ABB RobotStudio station: Project_Lab2.rsstnx

Station Project1 (saved by RobotStudio 25.1.11167.1)
Controller Controller_Lab2
  mechanical unit ROB_1: IRB140_6_81_C_03, 6 joints, base frame (0, 0, 0) mm
Layout (positions relative to the parent item):
  - IRB140_6_81_C_03 [mechanism, from %ABB.RobotStudio.Models.IRB140%\IRB140_6_81_C_G_03.rslib] at (0, 0, 0) mm; joint values [-0.0202, 0.226, 0.2165, 0.0425, 0.3433, -0.0544] (rad or m)
  - Marcador_2 [mechanism, from Project_Lab2\Marcador.rslib] at (539.94, -10, 494.18) mm, rotated rx -180 ry 45 rz -180 deg
  - Pastel [part] at (500, 0, 250) mm, rotated rx 0 ry 0 rz -90 deg, size 272 x 195 x 20 mm
Attachment: Marcador_2 is attached to IRB140_6_81_C_03 / Link6
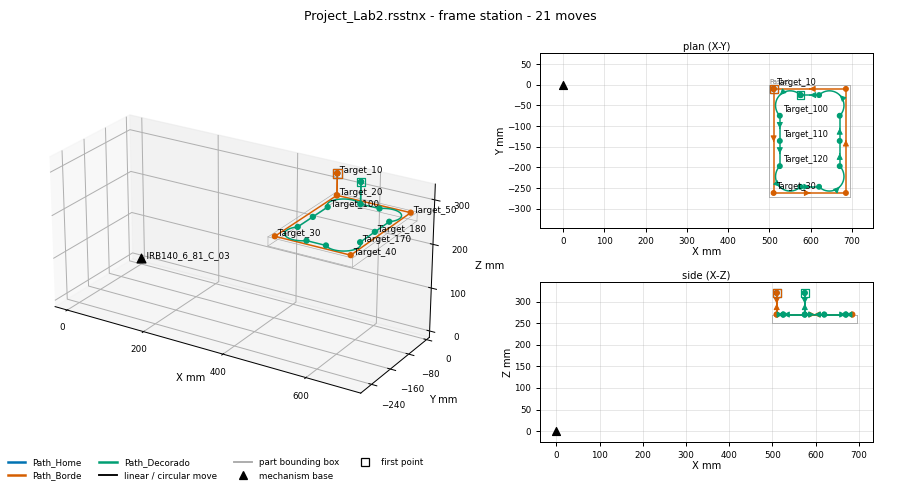
[picture p0: tool path of Project_Lab2.rsstnx in frame station, 21 of 21 moves have a stored position in this frame; points joined in program order, loops and branches not executed]
Targets, tools, work objects and paths stored in the station, written as RAPID:
! task T_ROB1
MODULE CalibData
  PERS tooldata TCP_Marcador:=[TRUE,[[144.332,0,101.99],[0.866025404,0,0.5,0]],[1,[0,0,1],[1,0,0,0],0,0,0]];
  TASK PERS wobjdata Workobject_pastel:=[FALSE,TRUE,"",[[500,0,250],[0.707106781,0,0,-0.707106781]],[[0,0,0],[1,0,0,0]]];
ENDMODULE

! task T_ROB1
MODULE Module1
  CONST robtarget Target_10:=[[10,10,70],[0.092295955,0.701057385,-0.701057385,0.092295955],[0,0,0,0],[9E+09,9E+09,9E+09,9E+09,9E+09,9E+09]];
  CONST robtarget Target_20:=[[10,10,20],[0.092295955,0.701057385,-0.701057385,0.092295955],[0,0,0,0],[9E+09,9E+09,9E+09,9E+09,9E+09,9E+09]];
  CONST robtarget Target_30:=[[262,10,20],[0.092295955,0.701057385,-0.701057385,0.092295955],[0,0,0,0],[9E+09,9E+09,9E+09,9E+09,9E+09,9E+09]];
  CONST robtarget Target_40:=[[262,185,20],[0.092295955,0.701057385,-0.701057385,0.092295955],[0,0,0,0],[9E+09,9E+09,9E+09,9E+09,9E+09,9E+09]];
  CONST robtarget Target_50:=[[10,185,20],[0.092295955,0.701057385,-0.701057385,0.092295955],[0,0,0,0],[9E+09,9E+09,9E+09,9E+09,9E+09,9E+09]];
  CONST robtarget Target_60:=[[10,10,20],[0.092295955,0.701057385,-0.701057385,0.092295955],[0,0,0,0],[9E+09,9E+09,9E+09,9E+09,9E+09,9E+09]];
  CONST robtarget Target_70:=[[25,75,70],[0.092295955,0.701057385,-0.701057385,0.092295955],[-1,0,-1,0],[9E+09,9E+09,9E+09,9E+09,9E+09,9E+09]];
  CONST robtarget Target_80:=[[25,75,20],[0.092295955,0.701057385,-0.701057385,0.092295955],[-1,0,-1,0],[9E+09,9E+09,9E+09,9E+09,9E+09,9E+09]];
  CONST robtarget Target_90:=[[25,25,20],[0.092295955,0.701057385,-0.701057385,0.092295955],[-1,0,-1,0],[9E+09,9E+09,9E+09,9E+09,9E+09,9E+09]];
  CONST robtarget Target_100:=[[75,25,20],[0.092295955,0.701057385,-0.701057385,0.092295955],[-1,0,-1,0],[9E+09,9E+09,9E+09,9E+09,9E+09,9E+09]];
  CONST robtarget Target_110:=[[136,25,20],[0.092295955,0.701057385,-0.701057385,0.092295955],[-1,0,-1,0],[9E+09,9E+09,9E+09,9E+09,9E+09,9E+09]];
  CONST robtarget Target_120:=[[197,25,20],[0.092295955,0.701057385,-0.701057385,0.092295955],[-1,0,-1,0],[9E+09,9E+09,9E+09,9E+09,9E+09,9E+09]];
  CONST robtarget Target_130:=[[247,25,20],[0.092295955,0.701057385,-0.701057385,0.092295955],[-1,0,-1,0],[9E+09,9E+09,9E+09,9E+09,9E+09,9E+09]];
  CONST robtarget Target_140:=[[247,75,20],[0.092295955,0.701057385,-0.701057385,0.092295955],[-1,0,-1,0],[9E+09,9E+09,9E+09,9E+09,9E+09,9E+09]];
  CONST robtarget Target_150:=[[247,120,20],[0.092295955,0.701057385,-0.701057385,0.092295955],[-1,0,-1,0],[9E+09,9E+09,9E+09,9E+09,9E+09,9E+09]];
  CONST robtarget Target_160:=[[247,170,20],[0.092295955,0.701057385,-0.701057385,0.092295955],[-1,0,-1,0],[9E+09,9E+09,9E+09,9E+09,9E+09,9E+09]];
  CONST robtarget Target_170:=[[197,170,20],[0.092295955,0.701057385,-0.701057385,0.092295955],[-1,0,-1,0],[9E+09,9E+09,9E+09,9E+09,9E+09,9E+09]];
  CONST robtarget Target_180:=[[136,170,20],[0.092295955,0.701057385,-0.701057385,0.092295955],[-1,0,-1,0],[9E+09,9E+09,9E+09,9E+09,9E+09,9E+09]];
  CONST robtarget Target_190:=[[75,170,20],[0.092295955,0.701057385,-0.701057385,0.092295955],[-1,0,-1,0],[9E+09,9E+09,9E+09,9E+09,9E+09,9E+09]];
  CONST robtarget Target_200:=[[25,170,20],[0.092295955,0.701057385,-0.701057385,0.092295955],[-1,0,-1,0],[9E+09,9E+09,9E+09,9E+09,9E+09,9E+09]];
  CONST robtarget Target_210:=[[25,120,20],[0.092295955,0.701057385,-0.701057385,0.092295955],[-1,0,-1,0],[9E+09,9E+09,9E+09,9E+09,9E+09,9E+09]];
  CONST robtarget Target_220:=[[25,75,20],[0.092295955,0.701057385,-0.701057385,0.092295955],[-1,0,-1,0],[9E+09,9E+09,9E+09,9E+09,9E+09,9E+09]];
  CONST robtarget Target_230:=[[25,75,70],[0.092295955,0.701057385,-0.701057385,0.092295955],[0,0,0,0],[9E+09,9E+09,9E+09,9E+09,9E+09,9E+09]];
  PROC main()
    Path_Home;
    WaitTime 1.5;
    Path_Borde;
    WaitTime 1.5;
    Path_Decorado;
    WaitTime 1.5;
    Path_Home;
  ENDPROC
  PROC Path_Home()
    MoveJ Target_10,v60,z100,TCP_Marcador\WObj:=Workobject_pastel;
  ENDPROC
  PROC Path_Borde()
    MoveL Target_10,v100,z10,TCP_Marcador\WObj:=Workobject_pastel;
    MoveL Target_20,v60,z10,TCP_Marcador\WObj:=Workobject_pastel;
    MoveL Target_30,v60,z10,TCP_Marcador\WObj:=Workobject_pastel;
    MoveL Target_40,v60,z10,TCP_Marcador\WObj:=Workobject_pastel;
    MoveL Target_50,v60,z10,TCP_Marcador\WObj:=Workobject_pastel;
    MoveL Target_60,v60,z10,TCP_Marcador\WObj:=Workobject_pastel;
    MoveL Target_10,v100,z10,TCP_Marcador\WObj:=Workobject_pastel;
  ENDPROC
  PROC Path_Decorado()
    MoveL Target_70,v60,z10,TCP_Marcador\WObj:=Workobject_pastel;
    MoveL Target_80,v60,z10,TCP_Marcador\WObj:=Workobject_pastel;
    MoveC Target_90,Target_100,v60,z10,TCP_Marcador\WObj:=Workobject_pastel;
    MoveL Target_110,v60,z10,TCP_Marcador\WObj:=Workobject_pastel;
    MoveL Target_120,v60,z10,TCP_Marcador\WObj:=Workobject_pastel;
    MoveC Target_130,Target_140,v60,z10,TCP_Marcador\WObj:=Workobject_pastel;
    MoveL Target_150,v60,z10,TCP_Marcador\WObj:=Workobject_pastel;
    MoveC Target_160,Target_170,v60,z10,TCP_Marcador\WObj:=Workobject_pastel;
    MoveL Target_180,v60,z10,TCP_Marcador\WObj:=Workobject_pastel;
    MoveL Target_190,v60,z10,TCP_Marcador\WObj:=Workobject_pastel;
    MoveC Target_200,Target_210,v60,z10,TCP_Marcador\WObj:=Workobject_pastel;
    MoveL Target_220,v60,z10,TCP_Marcador\WObj:=Workobject_pastel;
    MoveL Target_230,v60,z10,TCP_Marcador\WObj:=Workobject_pastel;
  ENDPROC
ENDMODULE

